# EPICS alarm handler configuration: mps_database/bare/alarms/areas/mpln_unds_mp02.alhConfig
GROUP NULL MPLN:UNDS:MP02:1
$ALIAS MPS Link Node 210
$GUIDANCE
LTUH MPS
   Group Name: MPLN:UNDS:MP02:1
   Summary PV:  MPLN:UNDS:MP02:1:STATSUMY
$END
CHANNEL  MPLN:UNDS:MP02:1    MPLN:UNDS:MP02:1:MPS_EN_RBV		-----
CHANNEL  MPLN:UNDS:MP02:1    MPLN:UNDS:MP02:1:LC1_MODE_RBV		-----
